{attribute addProperty BoxType "EL4102--0000"}
{attribute addProperty Id "OutputAT %Q*INT162"}
{attribute addProperty CRC "2526907244"}
{attribute addProperty SizeInBites "16"}
{attribute addProperty SizeInBytes "2"}
TYPE Channel_969D8B6C :
STRUCT
	{attribute addProperty Name "Output"}
	Output AT %Q* : INT;
END_STRUCT
END_TYPE

(* stored: Version 1.2.0.0, ProductVersion 3.1.4024.9
   DUT Channel_969D8B6C: Id {0c305965-6775-4edf-b9ec-eba6d8ff65f0} *)
